Staubli VAL3: page_editTraj.pjx

--- page_editTraj.pjx ---
Parameters version=s7.6.1 stackSize=5000 millimeterUnit=true
Program file=buildList.pgx
Program file=changePoint.pgx
Program file=goTo.pgx
Program file=insertInstr.pgx
Program file=listAdd.pgx
Program file=loadEditTraj.pgx
Program file=loadPage.pgx
Program file=main.pgx
Program file=onBackEvent.pgx
Program file=onEnterEvent.pgx
Program file=onExit.pgx
Program file=onF1Event.pgx
Program file=onF2Event.pgx
Program file=onF3Event.pgx
Program file=onF4Event.pgx
Program file=onF5Event.pgx
Program file=onF6Event.pgx
Program file=onF7Event.pgx
Program file=onF8Event.pgx
Program file=onSpaceEvent.pgx
Program file=onStart.pgx
Program file=refresh.pgx
Program file=refreshDynamic.pgx
Program file=refreshStatic.pgx
Program file=saveIt.pgx
Program file=selectItem.pgx
Program file=setAllAccel.pgx
Program file=setAllBlend.pgx
Program file=setAllSpeed.pgx
Program file=showPoint.pgx
Program file=showStatus.pgx
Program file=unSelectItem.pgx
Data file=page_editTraj.dtx
Library alias=use path=Disk://kernel/userPage/userPage.pjx
Library alias=language path=Disk://kernel/language/language.pjx
Library alias=saveData path=Disk://saveData/saveData.pjx
Library alias=trajType path=Disk://..//templates/trajectory/trajectory.pjx
Library alias=events path=Disk://..//templates/instruction/instruction.pjx
Library alias=tcp path=Disk://kernel/tool/tool.pjx
Library alias=page path=Disk://kernel/template/page/page.pjx
Library alias=cycleStatus path=Disk://cycleStatus/cycleStatus.pjx
Library alias=saveInOut path=Disk://saveInputOutput/saveInputOutput.pjx
Type name=TrajectoryItem path=Disk://kernel/template/TrajectoryItem/TrajectoryItem.pjx
Type name=InstrItem path=Disk://kernel/template/InstrItem/InstrItem.pjx
Type name=FrameItem path=Disk://kernel/template/FrameItem/FrameItem.pjx

--- page_editTraj.dtx ---
bool bButton[8]
  [0] = true
  [1] = true
  [2] = true
  [4] = true
  [5] = true
  [6] = true
  [7] = true
bool bExit
bool bLarge
bool bShowStatus
bool bTrigger
num nClockStatus = 962.397
num nIndex
num nIndexItem
num nKey
num nOldIndex
public num nPage
num nRefresh = 1149.353
num nSelected = -1
num nTime = 1
num nUserItem = 6
num nView
string sAction[3]
string sEvent = "Name: > appro"
public string sItems = "pick"
string sList[17]
  [0] = "Name: > appro"
  [1] = "appro   X > 0   "
  [2] = "appro   Y > 0   "
  [3] = "appro   Z > -50   "
  [4] = "appro  RX > 0   "
  [5] = "appro  RY > 0   "
  [6] = "appro  RZ > 0   "
  [7] = "MoveType > Linear"
  [8] = "Speed    > 1000 mm/s"
  [9] = "Accelerat> 100 %"
  [10] = "Stop  [ ]> "
  [11] = "Blend [x]> 30 mm"
  [12] = "Tool  [ ]>    "
  [13] = "Action1>  "
  [14] = "Action2>  "
  [15] = "Action3>  "
  [16] = "Anticipation > 0 mm"
string sListUser[6]
  [0] = "appro   X > 0   "
  [1] = "appro   Y > 0   "
  [2] = "appro   Z > -50   "
  [3] = "appro  RX > 0   "
  [4] = "appro  RY > 0   "
  [5] = "appro  RZ > 0   "
string sMenu[8]
  [0] = "Here"
  [1] = "Align"
  [2] = "Tool"
  [4] = "Motion"
  [5] = "Delete"
  [6] = "Insert"
  [7] = "Save"
string sMenu8[8]
string sMenuUser[8]
  [0] = "Here"
  [1] = "Align"
  [2] = "Tool"
string sMessage[2]
  [0] = "ON"
  [1] = "OFF"
string sOldListUser
string sTrajName = "pick"
frame fFather = {fatherId=world[0]}

--- main.pgx ---
public program main()
  local bool l_bSave
  local bool l_bOverRide
  local num l_nSize
  local bool l_bUnreached
  local string l_sMessage
begin
  // INIT
  call onStart()
  // LOOP UNTIL nKey=255
  do
    // GOTO
    call goTo(nIndexItem,l_bUnreached)
    if l_bUnreached
      // show the message out of range
      call language:message(l_sMessage,-5)
      call use:timerDialog(l_sMessage,1)
      l_bUnreached=false
    endIf
    //
    call refresh()
    nKey=getKey()
    call use:listevent(nKey,nIndex,sEvent)
    nView=use:nView
    // get Size
    call trajType:getSizeItem(false,l_nSize)
    //
    // OVERRIDE NORMAL FUNCTIONALITY-> POLYMORPHISM
    //
    if nKey>=271 and nKey<=278
      if sMenuUser[nKey-271]!=""
        call trajType:onFunctionEdit(nIndexItem,sEvent,nKey)
        l_bOverRide=true
        l_bSave=true
        call buildList()
      endIf
    endIf
    //
    // OVERRIDE ON ENTER EVENT -> POLYMORPHISM
    //
    if !l_bOverRide
      switch nKey
        case 264
          // left
          if nIndexItem>0
            nIndexItem=nIndexItem-1
            call buildList()
          endIf
        break
        case 268
          // right
          if nIndexItem<(l_nSize-1)
            nIndexItem=nIndexItem+1
            call buildList()
          endIf
        break
        case 259
          // TAB
          bLarge=!bLarge
          call use:setView(bLarge)
        break
        case 32
          call onSpaceEvent(l_bSave)
        break
        case 263
          call onBackEvent(l_bSave)
        break
        case 271
          call onF1Event()
        break
        case 272
          call onF2Event()
        break
        case 273
          call onF3Event()
        break
        case 274
          // Blend
          call onF4Event(l_bSave)
        break
        case 275
          // Speed
          call onF5Event(l_bSave)
        break
        case 276
          // Delete
          call onF6Event(l_bSave)
        break
        case 277
          // Insert
          call onF7Event(l_bSave)
        break
        case 278
          // SAVE
          call onF8Event(l_bSave)
        break
        case 270
          // GO EDIT POINT
          call onEnterEvent(l_bSave)
        break
      endSwitch
    endIf
    l_bOverRide=false
    if nKey==255
      // on Exit
      call onExit(l_bSave)
    endIf
    // release
    delay(0)
  until bExit
  // reset the bit
  bExit=false
end

--- buildList.pgx ---
program buildList()
  local num l_nSize
  local num i
  local string l_sInstruction
  local string l_sMessage
  local string l_sTemp
  local string l_sEmpty
  local TrajectoryItem l_tTraj
  local string l_sData
  local string l_sType
begin
  // INIT the list
  l_sEmpty=""
  call use:stringCopy(l_sEmpty,sList)
  // get all the field
  call trajType:getSizeItem(false,l_nSize)
  call trajType:getTrajItem(l_tTraj,nIndexItem)
  //
  // make the list
  //
  // the name
  call language:message(l_sMessage,21)
  call listAdd(l_sMessage+"> "+l_tTraj.comment)
  if find(l_tTraj.comment,"@")==-1
    // insert the user function if NOT @LINK
    call trajType:getListItem(sListUser,nIndexItem)
    if sListUser!=""
      for i=0 to size(sListUser)-1
        call listAdd(sListUser[i])
      endFor
      nUserItem=size(sListUser)
    else
      nUserItem=0
    endIf
    // check the size for the line underline
    if size(sListUser)!=size(sOldListUser) and sOldListUser!=""
      nSelected=nIndex+(size(sListUser)-size(sOldListUser))
      // copy it
      call use:stringCopy(sListUser,sOldListUser)
      use:bUseRefresh=true
    else
      nSelected=-1
    endIf
  else
    // empty it
    call use:stringCopy(l_sEmpty,sListUser)
    nUserItem=0
    nSelected=nIndex
  endIf
  // the movetype
  switch l_tTraj.moveType
    case 0
      // JOINT
      call language:message(l_sTemp,164)
      call language:message(l_sMessage,157)
      call use:strfill(l_sMessage,9,l_sMessage)
      call listAdd(l_sMessage+"> "+l_sTemp)
      call language:message(l_sMessage,158)
      call use:strfill(l_sMessage,9,l_sMessage)
      call listAdd(l_sMessage+"> "+toString("",l_tTraj.nom_speed.vel)+" %")
    break
    case 1
      //LINEAR
      call language:message(l_sTemp,165)
      call language:message(l_sMessage,157)
      call use:strfill(l_sMessage,9,l_sMessage)
      call listAdd(l_sMessage+"> "+l_sTemp)
      call language:message(l_sMessage,158)
      call use:strfill(l_sMessage,9,l_sMessage)
      call listAdd(l_sMessage+"> "+toString("",l_tTraj.nom_speed.tvel)+" mm/s")
    break
    case 2
      //  CIRCULAR
      call language:message(l_sTemp,166)
      call language:message(l_sMessage,157)
      call use:strfill(l_sMessage,9,l_sMessage)
      call listAdd(l_sMessage+"> "+l_sTemp)
      call language:message(l_sMessage,158)
      call use:strfill(l_sMessage,9,l_sMessage)
      call listAdd(l_sMessage+"> "+toString("",l_tTraj.nom_speed.tvel)+" mm/s")
    break
  endSwitch
  // ACCELERATION
  call language:message(l_sMessage,159)
  call use:strfill(l_sMessage,9,l_sMessage)
  call listAdd(l_sMessage+"> "+toString("",l_tTraj.nom_speed.accel)+" %")
  // STOP
  call use:showBoolStatus(l_tTraj.toStop,l_sTemp)
  call language:message(l_sMessage,174)
  call use:strfill(l_sMessage,6,l_sMessage)
  l_sMessage=l_sMessage+l_sTemp
  if l_tTraj.toStop
    // STOP
    if round(l_tTraj.nStop)!=l_tTraj.nStop
      l_sTemp=toString(".2",l_tTraj.nStop)+" sec"
    else
      l_sTemp=toString("",l_tTraj.nStop)+" sec"
    endIf
  else
    // NO STOP
    l_sTemp=""
  endIf
  call listAdd(l_sMessage+"> "+l_sTemp)
  // BLEND
  if l_tTraj.nom_speed.blend==off
    l_sTemp="[ ]> "
  else
    if l_tTraj.nom_speed.blend==joint
      l_sTemp="[x]> "+toString("",l_tTraj.nom_speed.leave)+" mm"
    endIf
  endIf
  call language:message(l_sMessage,175)
  call use:strfill(l_sMessage,6,l_sMessage)
  call listAdd(l_sMessage+l_sTemp)
  // TCP ON OFF
  call language:message(l_sMessage,123)
  call use:strfill(l_sMessage,6,l_sMessage)
  switch l_tTraj.nTcpAction
    case 1
      l_sTemp="[x]> ON "
    break
    case 2
      l_sTemp="[x]> OFF"
    break
    default
      l_sTemp="[ ]>    "
    break
  endSwitch
  call listAdd(l_sMessage+l_sTemp)
  // INSTRUCTION
  call language:message(l_sMessage,176)
  // copy all
  for i=0 to size(l_tTraj.iInstr)-1
    l_sData=l_tTraj.iInstr[i].sData
    l_sType=l_tTraj.iInstr[i].sType
    call saveInOut:replaceIO(l_sData,l_sType,l_sData)
    call listAdd(l_sMessage+toString("1",i+1)+"> "+l_sType+" "+l_sData)
  endFor
  // DISTANCE
  call language:message(l_sMessage,177)
  call listAdd(l_sMessage+" > "+toString("",l_tTraj.distance)+" mm")
  // update
  use:bUseRefresh=true
end

--- changePoint.pgx ---
program changePoint(num x_nIndex)
  local num i
  local string l_sMessage[3]
  local num l_nLocal
  local bool l_bOk
  local num l_nStop
  local string l_sButton[2]
  local string l_sEmpty
  local TrajectoryItem l_tTraj
  local InstrItem l_iInstr
  local string l_sItem
  local string l_sData
  local string l_sPath
begin
  //
  // Init and save the right side of the string starting from ">"
  //
  logMsg("[KERNEL] INTERFACE:Change Point: "+sEvent+" item: "+toString("",nIndexItem))
  //i=find(sEvent,">")+1
  call use:findPos(sEvent,">",i)
  i=i+1
  //
  if i!=-1
    //
    //  There are 10 fields,
    //
    call trajType:getTrajItem(l_tTraj,nIndexItem)
    // clean the line
    call use:listcursor(use:nView,false)
    l_sEmpty=""
    switch x_nIndex
      case 0
        //
        //  comment for the point
        //
        // read the name
        call use:read(i+40-use:nBottomX,use:nView+1,l_tTraj.comment,10,false)
      break
      case 1
        //
        //  change the movetype (0->Joint, 1->Linear, 2->Circle)
        //
        // JOINT
        if trajType:bMoveType[0]
          // normaly with joint can be also linear and circle
          call language:message(l_sMessage,164)
          call language:message(l_sMessage[1],165)
          call language:message(l_sMessage[2],166)
          if trajType:bMoveType[1]
            l_sMessage=l_sMessage+","+l_sMessage[1]
          endIf
          if trajType:bMoveType[2] and nIndexItem!=0
            l_sMessage=l_sMessage+","+l_sMessage[2]
          endIf
        else
          // only linear
          if trajType:bMoveType[1]
            l_sMessage=l_sMessage
          endIf
        endIf
        // compose the string
        call use:stringToArray(l_sMessage,sMessage)
        // look for multiple istance
        if size(sMessage)>1
          //
          l_nLocal=l_tTraj.moveType
          call use:changeValue(l_tTraj.moveType,0,0,i+40-use:nBottomX,use:nView+1,sMessage)
          if l_nLocal!=l_tTraj.moveType
            switch l_tTraj.moveType
              case 0
                if l_tTraj.nom_speed.tvel!=9999
                  l_tTraj.nom_speed.vel=(l_tTraj.nom_speed.tvel)/15
                  l_tTraj.nom_speed.tvel=9999
                endIf
              break
              case 1,2
                if l_tTraj.nom_speed.vel<450
                  l_tTraj.nom_speed.tvel=(l_tTraj.nom_speed.vel)*15
                  l_tTraj.nom_speed.vel=450
                endIf
              break
            endSwitch
            // update the line
            if l_nLocal==2 and nIndex>0 and nView>0
              // refresh the cursor
              nView=nView-1
              nIndex=nIndex-1
            else
              if l_tTraj.moveType==2
                // refresh the cursor
                nView=nView+1
                nIndex=nIndex+1
              endIf
            endIf
          endIf
        endIf
      break
      case 2
        //
        //  change the speed
        //
        if l_tTraj.moveType==0
          call use:changeValue(l_tTraj.nom_speed.vel,1,400,i+40-use:nBottomX,use:nView+1,l_sEmpty)
        else
          if l_tTraj.moveType==1 or l_tTraj.moveType==2
            call use:changeValue(l_tTraj.nom_speed.tvel,1,6000,i+40-use:nBottomX,use:nView+1,l_sEmpty)
          endIf
        endIf
      break
      case 3
        //
        //  change the acceleration
        //
        call use:changeValue(l_tTraj.nom_speed.accel,1,800,i+40-use:nBottomX,use:nView+1,l_sEmpty)
        l_tTraj.nom_speed.decel=l_tTraj.nom_speed.accel
      break
      case 4
        //
        //  put a stop, after the robot reach to the point
        //
        l_nLocal=l_tTraj.nStop
        call use:changeValue(l_nLocal,-1,100,i+40-use:nBottomX,use:nView+1,l_sEmpty)
        //
        if l_nLocal<0
          // no stop
          l_tTraj.toStop=false
          l_tTraj.nStop=0
        else
          // stop using time
          l_tTraj.toStop=true
          l_tTraj.nStop=l_nLocal
        endIf
      break
      case 5
        //
        //  set the blend (joint/off) for the point
        //
        l_nLocal=l_tTraj.nom_speed.leave
        call use:changeValue(l_nLocal,-1,400,i+40-use:nBottomX,use:nView+1,l_sEmpty)
        if l_nLocal<0
          l_tTraj.nom_speed.blend=off
        else
          l_tTraj.nom_speed.leave=l_tTraj.nom_speed.reach=l_nLocal
          l_tTraj.nom_speed.blend=joint
        endIf
      break
      case 6
        //
        // set TCP ON/OFF
        //
        // NB: 0>NONE 1>ON 2>OFF
        call use:stringToArray("ON,OFF",sMessage)
        if l_tTraj.nTcpAction!=0 and abs(l_tTraj.nTcpAction)<3
          // NOTE
          // use only absolute
          l_tTraj.nTcpAction=abs(l_tTraj.nTcpAction)-1
        else
          l_tTraj.nTcpAction=0
        endIf
        call use:changeValue(l_tTraj.nTcpAction,0,0,i+40-use:nBottomX,use:nView+1,sMessage)
        // give back increase by one
        l_tTraj.nTcpAction=l_tTraj.nTcpAction+1
      break
      case 7,8,9
        //
        //  Insert the instruction
        //
        // insert a new one
        if l_tTraj.iInstr[x_nIndex-7].sType!=""
          // show it
          if l_tTraj.iInstr[x_nIndex-7].sType=="OUT" or l_tTraj.iInstr[x_nIndex-7].sType=="IN" or l_tTraj.iInstr[x_nIndex-7].sType=="EMAP"
            popUpMsg(l_tTraj.iInstr[x_nIndex-7].sType+" "+l_tTraj.iInstr[x_nIndex-7].sData)
          else
            // update
            l_sItem=l_tTraj.iInstr[x_nIndex-7].sType
            l_sData=l_tTraj.iInstr[x_nIndex-7].sData
            call saveData:getPathInstr(l_sItem,l_sPath)
            events:libLoad(l_sPath)
            delay(0)
            call events:onEdit(l_sData)
            if l_sData!=""
              l_tTraj.iInstr[x_nIndex-7].sData=l_sData
            endIf
          endIf
        else
          // insert
          call insertInstr(l_iInstr)
          if l_iInstr.sData!=""
            l_tTraj.iInstr[x_nIndex-7]=l_iInstr
          endIf
        endIf
      break
      case 10
        //
        //  set the distance from the point where the call will be actived
        //
        call use:changeValue(l_tTraj.distance,-300,300,i+40-use:nBottomX,use:nView+1,l_sEmpty)
      break
    endSwitch
    //set and exit
    call trajType:setTrajItem(l_tTraj,nIndexItem)
  endIf
  //
  call use:nullKey(nKey)
end

--- goTo.pgx ---
program goTo(num x_nIndex, bool& x_bUnreached[])
  local bool l_bUnreached
  local num l_nIndexTool
  local tool l_tTool
  local TrajectoryItem l_tTraj
begin
//  if !cycleStatus:bCycle
//    if cycleStatus:nWorkingMode==1 and isPowered()
//      // check for the index
//      if nOldIndex!=x_nIndex or (cycleStatus:nWorkingStatus!=0 and cycleStatus:nWorkingStatus!=6)
//        if !isEmpty()
//          resetMotion()
//        endIf
//        if nOldIndex!=x_nIndex
//          nOldIndex=x_nIndex
//        endIf
//      else
//        if isEmpty() and cycleStatus:nWorkingStatus==0
//          // get the data to move
//          call trajType:getTool(l_nIndexTool)
//          call tcp:getTool(l_tTool,l_nIndexTool)
//          call trajType:getTrajItem(l_tTraj,x_nIndex)
//          //
//          // use a sTemp mdesc to set the blend off
//          //
//          l_tTraj.nom_speed.blend=off
//          call trajType:goTo(l_tTool,l_tTraj.nom_speed,l_tTraj.moveType,x_bUnreached,x_nIndex)
//          call showPoint()
//        endIf
//      endIf
//    else
//      if cycleStatus:nWorkingMode!=1
//        resetMotion()
//      endIf
//    endIf
//  endIf
end

--- insertInstr.pgx ---
program insertInstr(InstrItem& x_iInstr[])
  local num i
  local string l_sMessage
  local num l_nIndex
  local string l_sItem
  local string l_sPath
begin
  // create the list
  call use:setSizeList(15,0,15,11)
  call use:setView(false)
  call language:message(l_sMessage,35)
  call use:listcreate(l_sMessage)
  // insert the action on Point
  call use:listadd(saveData:sInstrOnPoint)
  call use:listupdate(0)
  // SELECT THE ITEM
  x_iInstr.sData=""
  do
    i=get()
    l_nIndex=0
    call use:listevent(i,l_nIndex,l_sItem)
  until i==255 or i==270
  // update
  x_iInstr.sType=l_sItem
  // update
  call saveData:getPathInstr(l_sItem,l_sPath)
  if l_sItem!="" and i==270
    events:libLoad(l_sPath)
    delay(0)
    call events:onInsert(l_sItem)
    x_iInstr.sData=l_sItem
  endIf
end

--- loadEditTraj.pgx ---
program loadEditTraj(string x_sName)
  local num i
  local num l_nIndex
  local string l_sPath
begin
  // load the traj type
  call saveData:getPathInstr(saveData:sTrajTypeUsing,l_sPath)
  i=trajType:libLoad(l_sPath)
  delay(0)
  if i!=0
    popUpMsg("error load traj type on START "+saveData:sTrajTypeUsing+toString("",i))
  endIf
  // save the name
  sTrajName=x_sName
end

--- loadPage.pgx ---
program loadPage(string x_sPage, string& x_sItems[])
// load the next page
  local num i
  local string l_sMessage
begin
  // look if the page libload is correct
  i=page:libLoad(x_sPage)
  delay(0)
  if i!=0
    logMsg("[KERNEL] INTERFACE:PAGE LIBLOAD "+x_sPage+" result "+toString("",i))
    call language:message(l_sMessage,-7)
    popUpMsg(l_sMessage+x_sPage+" ; "+toString("",i))
  else
    // copy all the field from x_sItems to the next page
    call use:stringCopy(x_sItems,page:sItems)
    call page:main()
    // copy BACK
    call use:stringCopy(page:sItems,x_sItems)
  endIf
end

--- onBackEvent.pgx ---
program onBackEvent(bool& x_bSave[] (dimensions=1))
  local num i
  local string l_sMessage[3]
  local num l_nLocal
  local bool l_bYes
  local string l_sAction[3]
  local num l_nIndex
  local string l_sButton[2]
  local TrajectoryItem l_tTraj
begin
  //
  // NB sEvent is the selected
  // element in the LIST
  //
  if nIndex!=0
    l_nIndex=nIndex-nUserItem
  else
    // change the name
    call changePoint(0)
  endIf
  if (l_nIndex)>0
    //
    //  There are 7 fields,
    //
    //
    call trajType:getTrajItem(l_tTraj,nIndexItem)
    switch l_nIndex
      case 1
        //
        //  change the movetype
        //
      break
      case 2
        //
        //  change the speed
        //
      break
      case 3
        //
        //  change the acceleration
        //
      break
      case 4
        //
        //  put a stop, after the robot reach to the point
        //
        // CLEAR THE STOP
        l_tTraj.toStop=false
      break
      case 5
        //
        //  set the blend (joint/off) for the point
        //
        l_tTraj.nom_speed.blend=off
      break
      case 6
        //
        // set TCP ON/OFF
        //
        // SET TCP OFF
        l_tTraj.nTcpAction=0
      break
      case 7,8,9
        //
        //  Delete the instruction
        //
        if l_tTraj.iInstr[l_nIndex-7].sType!=""
          call language:message(l_sMessage,171)
          call language:getYesNo(l_sButton)
          // ask the yes_no question
          call use:yes_no(l_sMessage,l_sButton,l_bYes)
          if l_bYes
            l_tTraj.iInstr[l_nIndex-7].sType=""
            l_tTraj.iInstr[l_nIndex-7].sData=""
          endIf
        endIf
      break
      case 10
        //
        //  set the distance from the point where the call will be actived
        //
        l_tTraj.distance=0
      break
    endSwitch
    //set and exit
    x_bSave=true
    call trajType:setTrajItem(l_tTraj,nIndexItem)
    call buildList()
  endIf
end

--- onEnterEvent.pgx ---
program onEnterEvent(bool& x_bSave (dimensions=1))
begin
  //
  // NB sEvent is the selected
  // element in the LIST
  //
  if nIndex==0
    // change the name
    call changePoint(0)
  else
    if (nIndex-nUserItem)>0
      // change the default value
      call changePoint(nIndex-nUserItem)
      x_bSave=true
    else
      // change the custom item
      call trajType:onEditItem(sEvent,nIndex-1,nIndexItem)
    endIf
  endIf
  x_bSave=true
  call buildList()
end

--- onExit.pgx ---
program onExit(bool& x_bSave[] (dimensions=1))
  local string l_sMessage
  local bool l_bYes
  local bool l_bCancel
  local string l_sButton[2]
begin
  // saveIt
  if x_bSave
    call language:message(l_sMessage,-1)
    call language:getYesNo(l_sButton)
    // ask the yes_no question
    call use:yes_no_cancel(l_sMessage,l_sButton,l_bYes,l_bCancel)
    if l_bYes
      call saveIt(x_bSave)
    endIf
    // look for the cancel button
    bExit=!l_bCancel
  else
    // exit frome the page
    bExit=true
  endIf
  // send Back
  if size(sItems)>1
    sItems[1]=toString("",nIndexItem)
  endIf
  // null key
  call use:nullKey(nKey)
  // reset the show status
  bShowStatus=false
  // resetMotion
  if !cycleStatus:bCycle
    resetMotion()
  endIf
end

--- onF1Event.pgx ---
program onF1Event()
begin
  // look if the bButton is enable
  if bButton[0]
    //
  endIf
end

--- onF4Event.pgx ---
program onF4Event(bool& x_bSave[] (dimensions=1))
  local string l_sMessage
  local num l_nActual
  local num l_nOldValue
  local num l_nX
  local num l_nY
begin
  // look if the bButton is enable
  if bButton[3]
    //
    //
    //
  endIf
end

--- onF5Event.pgx ---
program onF5Event(bool& x_bSave[])
  local string l_sMessage
  local num l_nActual
  local num l_nOldValue
  local num l_nMoveType
  local num l_nIndex
  local num l_nKey
  local string l_sEvent
  local TrajectoryItem l_tTraj
begin
  // look if the bButton is enable
  if bButton[4]
    //
    // build a little List to select speed accel blend
    //
    call use:clear(0,13)
    call use:type(21,13,sMenu[4])
    call use:setSizeList(17,8,12,3)
    call use:listcreate("")
    // speed
    call language:message(l_sMessage,158)
    call use:listadd(l_sMessage)
    // accel
    call language:message(l_sMessage,159)
    call use:listadd(l_sMessage)
    // blend
    call language:message(l_sMessage,175)
    call use:listadd(l_sMessage)
    //
    call use:listupdate(0)
    do
      l_nKey=get()
      call use:listevent(l_nKey,l_nIndex,l_sEvent)
    until l_nKey==270 or l_nKey==255
    if l_nKey==270
      // get the traj Item
      call trajType:getTrajItem(l_tTraj,nIndexItem)
      // switch case
      switch l_nIndex
        case 0
          //
          // change the speed
          //
          call language:message(l_sMessage,161)
          switch l_tTraj.moveType
            case 0
              // JOINT
              l_nActual=l_nOldValue=l_tTraj.nom_speed.vel
              call use:insertDialog(l_sMessage+" %",l_nActual,1,400)
            break
            case 1,2
              //LINEAR CIRCULAR
              l_nActual=l_nOldValue=l_tTraj.nom_speed.tvel
              call use:insertDialog(l_sMessage+" mm/sec ",l_nActual,1,6000)
            break
          endSwitch
          call setAllSpeed(l_nActual,l_nOldValue)
          logMsg("[VALTRAJ] INTERFACE:Change all speed from: "+toString("",l_nOldValue)+" to: "+toString("",l_nActual))
        break
        case 1
          //
          // CHANGE ALL THE ACCEL
          //
          call language:message(l_sMessage,162)
          l_nActual=l_nOldValue=l_tTraj.nom_speed.accel
          call use:insertDialog(l_sMessage,l_nActual,1,800)
          call setAllAccel(l_nActual,l_nOldValue)
          logMsg("[VALTRAJ] INTERFACE:Change all accel from: "+toString("",l_nOldValue)+" to: "+toString("",l_nActual))
        break
        case 2
          //
          // CHANGE ALL THE BLEND
          //
          call language:message(l_sMessage,178)
          l_nActual=l_nOldValue=l_tTraj.nom_speed.leave
          call use:insertDialog(l_sMessage,l_nActual,-1,400)
          call setAllBlend(l_nActual,l_nOldValue)
          logMsg("[VALTRAJ] INTERFACE:Change all blend from: "+toString("",l_nOldValue)+" to: "+toString("",l_nActual))
        break
      endSwitch
      // save and return
      x_bSave=true
      call buildList()
    endIf
  endIf
end

--- onF6Event.pgx ---
program onF6Event(bool& x_bSave[])
  local string l_sMessage
  local bool l_bYes
  local num l_nSize
  local num l_nFound
  local string l_sEvent
  local string l_sButton[2]
  local num l_nItem
begin
  // look if the bButton is enable
  if bButton[5]
    //
    // DELETE
    //
    call language:message(l_sMessage,80)
    call language:getYesNo(l_sButton)
    // ask the yes_no question
    call use:yes_no(l_sMessage,l_sButton,l_bYes)
    if l_bYes
      l_nItem=nIndexItem
      call trajType:getSizeItem(false,l_nSize)
      if l_nSize>1
        call trajType:deleteItem(nIndexItem)
        if nIndexItem>0
          nIndexItem=nIndexItem-1
        else
          nIndexItem=l_nItem
        endIf
        //refresh
        call buildList()
        use:bUseRefresh=true
      endIf
    endIf
    x_bSave=true
  endIf
end

--- onF7Event.pgx ---
program onF7Event(bool& x_bSave[] (dimensions=1))
  local TrajectoryItem l_tTraj
  local num l_nItem
begin
  // look if the bButton is enable
  if bButton[6]
    //
    // insert
    l_nItem=nIndexItem
    // insert the default value
    call trajType:insertItem(nIndexItem,nIndexItem+1)
    call trajType:getTrajItem(l_tTraj,nIndexItem)
    l_tTraj.comment=""
    l_tTraj.toStop=false
    call trajType:setTrajItem(l_tTraj,nIndexItem+1)
    nIndexItem=nIndexItem+1
    // rebuild list
    call buildList()
    x_bSave=true
    //refresh
    call buildList()
    use:bUseRefresh=true
  endIf
end

--- onF8Event.pgx ---
program onF8Event(bool& x_bSave[] (dimensions=1))
  local num i
begin
  // look if the bButton is enable
  if bButton[7]
    //
    call saveIt(x_bSave)
  endIf
end

--- onSpaceEvent.pgx ---
program onSpaceEvent(bool& x_bSave[])
  local num i
  local string l_sMessage[3]
  local num l_nLocal
  local bool l_bYes
  local string l_sAction[3]
  local num l_nIndex
  local TrajectoryItem l_tTraj
  local bool l_bStop
begin
  //
  // NB sEvent is the selected
  // element in the LIST
  //
  l_nIndex=nIndex-nUserItem
  if (nIndex-nUserItem)>0
    //
    //  There are 7 fields,
    //
    //
    call trajType:getTrajItem(l_tTraj,nIndexItem)
    switch l_nIndex
      case 0
        //
        //  comment for the point
        //
      break
      case 1
        //
        //  change the movetype
        //
      break
      case 2
        //
        //  change the speed
        //
      break
      case 3
        //
        //  change the acceleration
        //
      break
      case 4
        //
        //  put a stop, after the robot reach to the point
        //
        l_tTraj.toStop=!l_tTraj.toStop
      break
      case 5
        //
        //  set the blend (joint/off) for the point
        //
        if l_tTraj.nom_speed.blend==off
          l_tTraj.nom_speed.blend=joint
        else
          l_tTraj.nom_speed.blend=off
        endIf
      break
      case 6
        //
        // set TCP ON/OFF
        //
        if l_tTraj.nTcpAction!=0
          l_tTraj.nTcpAction=-l_tTraj.nTcpAction
        else
          // ON by default
          l_tTraj.nTcpAction=1
        endIf
      break
      case 7,8,9
        //
        //  Insert the instruction
        //
      break
      case 10
        //
        //  set the distance from the point where the call will be actived
        //
      break
    endSwitch
    //set and exit
    call trajType:setTrajItem(l_tTraj,nIndexItem)
    x_bSave=true
    call buildList()
  endIf
end

--- onStart.pgx ---
program onStart()
  local num i
  local num l_nIndex
  local bool l_bOk
begin
  // INIT
  sTrajName=sItems
  nView=0
  nIndex=0
  bExit=false
  link(fFather,world)
  call trajType:getFrame(fFather,false)
  // set the index
  l_bOk=true
  if size(sItems)>1 and sItems[1]!=""
    toNum(sItems[1],nIndexItem,l_bOk)
  else
    nIndexItem=0
  endIf
  // empty the userMenu
  for i=0 to size(sMenuUser)-1
    sMenuUser[i]=""
  endFor
  // load the traj type
  call loadEditTraj(sItems)
  //endIf
  //
  // logMsg
  logMsg("[KERNEL] INTERFACE:PAGE Edit TRAJ")
  // reset the Key pressure
  call use:nullKey(nKey)
  // define the list
  call buildList()
  //
end

--- refresh.pgx ---
program refresh()
// // page refresh
begin
  if !use:bShowDialog and !cycleStatus:bShowMessage
    //
    // refresh the static message
    if (nKey>=270 and nKey<=278) or (nKey==264 or nKey==268) or (use:bUseRefresh and !bShowStatus)
      call refreshStatic()
      call refreshDynamic()
    else
      if !bShowStatus
        // refresh the Dynamic message
        if abs(clock()-nRefresh)>nTime
          call refreshDynamic()
        endIf
      endIf
    endIf
  endIf
  //
  call showStatus()
end

--- refreshDynamic.pgx ---
program refreshDynamic()
begin
  // DO NOT CHANGE
  nRefresh=clock()
  use:bUseRefresh=false
  call showPoint()
  //
  // ADD HERE
  //
end

--- refreshStatic.pgx ---
program refreshStatic()
  local string l_sMenu
  local num i
  local string l_sInstruction
  local num l_nSize
  local string l_sMessage
  local mdesc l_mDesc
  local num l_nTcpAction
  local string l_sName
  local string l_sEmpty
  local bool l_bStop
  local num l_nEmpty
  local num l_nIndexTool
  local TrajectoryItem l_tTraj
  local string l_sType
  local string l_sData
begin
  cls()
  //
  // set the view of the page..
  //
  // SET THE PAGE NUMBER
  use:nPage=100000
  // USE <>PROFILE for <>PAGE
  use:nPage=use:nPage+abs(limit(saveData:mode,0,2)-2)
  // load the menu page
  if saveData:language!="japanese"
    // SET THE VIEW OF THE PAGE
    call language:page(l_sMessage,use:nPage)
    // define the menu
    call use:stringToArray(l_sMessage,sMenu)
  else
    // japanese use the array for the menu
    call language:page(sMenu8,use:nPage)
    call use:stringCopy(sMenu8,sMenu)
  endIf
  //
  // polymorphism
  //
  // get the user Menu or special one
  call trajType:getFunctionEdit(sMenuUser)
  // OVERRIDE
  for i=0 to size(sMenuUser)-1
    if sMenuUser[i]!=""
      sMenu[i]=sMenuUser[i]
    endIf
  endFor
  // check for the here if not in cycle
  if cycleStatus:bCycle or cycleStatus:bSimulation
    sMenu[0]=""
  endIf
  // remove the insert delete in this page
  sMenu[5]=sMenu[6]=""
  if saveData:language!="japanese"
    // set the menu
    call use:setMenu(sMenu,true,3)
  else
    // set the menu
    call use:setMenu(sMenu,false,3)
  endIf
  call use:getMenu(sMenu,bButton)
  //
  // CREATE THE LIST
  //
  // define your list size for default
  // get the nSize
  call trajType:getSizeItem(false,l_nSize)
  call use:setSizeList(19,0,19,10)
  call use:setView(bLarge)
  // show the title...
  l_sName=sTrajName
  if !bLarge and len(sTrajName)>12
    // as japanese told us
    l_sName=left(sTrajName,9)+"¬"+right(sTrajName,2)
  endIf
  call use:listcreate(l_sName+" "+toString("3",nIndexItem+1)+"/"+toString("3",l_nSize))
  //
  call use:listadd(sList)
  //
  // refresh the cursor
  use:nView=nView
  // refresh the list
  call use:selectNewField(nSelected,nIndex,nView)
  // show the instruction
  l_sEmpty=""
  l_bStop=false
  l_nEmpty=0
  call trajType:getTrajItem(l_tTraj,nIndexItem)
  // select the action
  switch l_tTraj.nTcpAction
    case 1
      l_sInstruction="[ON],"
    break
    case 2
      l_sInstruction="[OFF],"
    break
    default
    break
  endSwitch
  l_sType=l_tTraj.iInstr[0].sType
  l_sData=l_tTraj.iInstr[0].sData
  call saveInOut:replaceIO(l_sData,l_sType,l_sData)
  l_sInstruction=l_sInstruction+l_sType+" "+l_sData
  for i=1 to size(l_tTraj.iInstr)-1
    if l_tTraj.iInstr[i].sType!=""
      l_sType=l_tTraj.iInstr[i].sType
      l_sData=l_tTraj.iInstr[i].sData
      call saveInOut:replaceIO(l_sData,l_sType,l_sData)
      l_sInstruction=l_sInstruction+","+l_sType+" "+l_sData
    endIf
  endFor
  call use:typeLen(0,12,l_sInstruction,40)
  // TOOL - FRAME
  if !bLarge
    call trajType:getTool(i)
    call language:message(l_sMessage,124)
    call tcp:getName(l_sName,i)
    call use:type(0,0,l_sMessage+":"+toString("",i)+" "+l_sName)
    call trajType:getFrameId(i)
    call language:message(l_sMessage,124)
    l_sName=saveData:fFrameItem[i].sName
    call use:type(0,1,"Frame:"+toString("",i)+" "+l_sName)
  endIf
end

--- saveIt.pgx ---
program saveIt(bool& x_bSave[] (dimensions=1))
  local string l_sMessage
  local num l_nResult
  local string l_sResult
begin
  // unselect ALL
  call unSelectItem()
  // do the onSave trajtype
  l_sResult=""
  call trajType:onSave(l_sResult)
  //
  if l_nResult==0
    logMsg("[KERNEL] INTERFACE:Save the trajectory "+saveData:sTrajTypeUsing+": "+sTrajName)
    x_bSave=false
    call language:message(l_sMessage,-4)
    call use:timerDialog(l_sMessage,1)
  else
    popUpMsg("Save code error "+toString("",l_nResult))
  endIf
end

--- selectItem.pgx ---
public program selectItem(num x_nIndex (dimensions=1))
  local string l_sItem
  local TrajectoryItem l_tTraj
begin
  //
  // select or unselect one item
  //
  call trajType:getTrajItem(l_tTraj,x_nIndex)
  // check for the selected flag
  if find(l_tTraj.comment,"#")==-1
    l_tTraj.comment="#"+l_tTraj.comment
  else
    l_tTraj.comment=right(l_tTraj.comment,len(l_tTraj.comment)-1)
  endIf
  // set it
  call trajType:setTrajItem(l_tTraj,x_nIndex)
end

--- setAllAccel.pgx ---
public program setAllAccel(num x_nNewValue (dimensions=1), num x_nOldValue (dimensions=1))
  local num i
  local num l_nSize
  local TrajectoryItem l_tTraj
begin
  //
  // change all the accel(equal at newValue)to the newValue
  //
  if x_nNewValue!=x_nOldValue
    call trajType:getSizeItem(false,l_nSize)
    // scan it
    for i=0 to (l_nSize-1)
      // get it
      call trajType:getTrajItem(l_tTraj,i)
      // check if is OK
      if l_tTraj.nom_speed.accel==x_nOldValue
        l_tTraj.nom_speed.accel=l_tTraj.nom_speed.decel=x_nNewValue
      endIf
      // set IT
      call trajType:setTrajItem(l_tTraj,i)
    endFor
  endIf
end

--- setAllBlend.pgx ---
public program setAllBlend(num x_nNewValue, num x_nOldValue)
  local num i
  local num l_nSize
  local TrajectoryItem l_tTraj
begin
  // check if is OK
  if x_nNewValue!=x_nOldValue
    // get the size
    call trajType:getSizeItem(false,l_nSize)
    for i=0 to (l_nSize-1)
      // get it
      call trajType:getTrajItem(l_tTraj,i)
      // check it
      if l_tTraj.nom_speed.leave==x_nOldValue or (l_tTraj.nom_speed.blend==off and x_nOldValue==-1)
        if x_nNewValue<0
          l_tTraj.nom_speed.blend=off
        else
          l_tTraj.nom_speed.leave=l_tTraj.nom_speed.reach=x_nNewValue
          l_tTraj.nom_speed.blend=joint
        endIf
      endIf
      // set it
      call trajType:setTrajItem(l_tTraj,i)
    endFor
  endIf
end

--- setAllSpeed.pgx ---
program setAllSpeed(num x_nNewValue (dimensions=1), num x_nOldValue (dimensions=1))
  local num i
  local num l_nSize
  local TrajectoryItem l_tTraj
begin
  // change all the speed
  if x_nNewValue!=x_nOldValue
    call trajType:getSizeItem(false,l_nSize)
    // scan it
    for i=0 to (l_nSize-1)
      // get the trajitem
      call trajType:getTrajItem(l_tTraj,i)
      // JOINT MOVEMENT
      if (l_tTraj.moveType==0) and (x_nOldValue==l_tTraj.nom_speed.vel)
        l_tTraj.nom_speed.vel=x_nNewValue
        // LINEAR MOVEMENT
      elseIf (l_tTraj.moveType==1 or l_tTraj.moveType==2) and (x_nOldValue==l_tTraj.nom_speed.tvel)
        l_tTraj.nom_speed.tvel=x_nNewValue
      endIf
      // set the trajItem
      call trajType:setTrajItem(l_tTraj,i)
    endFor
  endIf
end

--- showPoint.pgx ---
program showPoint()
  local point l_pPoint[2]
  local num l_nIndexTool
  local tool l_tTool
  local point l_pHere
  local num i
  local joint l_jHere
begin
  // check for the @ position and the ! position
  call trajType:getPoint(l_pPoint,false,nIndexItem)
  call trajType:getTool(l_nIndexTool)
  call tcp:getTool(l_tTool,l_nIndexTool)
  l_pHere=here(l_tTool,fFather)
  if isEmpty() and distance(l_pHere.trsf,position(l_pPoint,fFather))<0.1
    call use:type(use:nTopX,use:nTopY+1,"@")
  elseIf position(l_pPoint,fFather)=={0,0,0,0,0,0}
    call use:type(use:nTopX,use:nTopY+1,"0")
  elseIf distance(position(l_pPoint,fFather),l_pHere.trsf)<10
    call use:type(use:nTopX,use:nTopY+1,"~")
  elseIf !pointToJoint(l_tTool,l_jHere,l_pPoint,l_jHere)
    call use:type(use:nTopX,use:nTopY+1,"!")
  else
    call use:type(use:nTopX,use:nTopY+1,"│")
  endIf
end

--- showStatus.pgx ---
program showStatus()
  local joint l_jHere
  local point l_pHere
  local string l_sMessage[2]
  local tool l_tTool
  local num l_nIndexTool
begin
  //
  // show an dialog box with
  // the current Joint/cartesian position
  //
  call trajType:getTool(l_nIndexTool)
  call tcp:getTool(l_tTool,l_nIndexTool)
  if cycleStatus:nWorkingStatus>1 and cycleStatus:nWorkingStatus<5 and cycleStatus:nWorkingMode==1
    // set a timer of x second then the message disappear ..
    if !bTrigger
      nClockStatus=clock()
      bTrigger=true
      bShowStatus=true
    endIf
    if clock()-nClockStatus<saveData:nTimeDialog
      if cycleStatus:nWorkingStatus==2
        l_jHere=herej()
        l_sMessage="J1:"+toString("7.1",l_jHere.j1)
        l_sMessage=l_sMessage+"  J2:"+toString("7.1",l_jHere.j2)
        l_sMessage=l_sMessage+"  J3:"+toString("7.1",l_jHere.j3)+"#"
        l_sMessage=l_sMessage+"J4:"+toString("7.1",l_jHere.j4)
        l_sMessage=l_sMessage+"  J5:"+toString("7.1",l_jHere.j5)
        l_sMessage=l_sMessage+"  J6:"+toString("7.1",l_jHere.j6)
      else
        l_pHere=here(l_tTool,fFather)
        l_sMessage="X :"+toString("7.1",l_pHere.trsf.x)
        l_sMessage=l_sMessage+"  Y :"+toString("7.1",l_pHere.trsf.y)
        l_sMessage=l_sMessage+"  Z :"+toString("7.1",l_pHere.trsf.z)+"#"
        l_sMessage=l_sMessage+"RX:"+toString("7.1",l_pHere.trsf.rx)
        l_sMessage=l_sMessage+"  RY:"+toString("7.1",l_pHere.trsf.ry)
        l_sMessage=l_sMessage+"  RZ:"+toString("7.1",l_pHere.trsf.rz)
      endIf
      call use:timerDialog(l_sMessage,0)
    else
      // disable it
      bShowStatus=false
    endIf
  else
    // reset it
    if bTrigger and !cycleStatus:bCycle
      resetMotion()
      call showPoint()
    endIf
    bTrigger=false
    bShowStatus=false
  endIf
end

--- unSelectItem.pgx ---
program unSelectItem()
  local string l_sEvent
  local num i
  local num l_nSize
  local TrajectoryItem l_tTraj
begin
  // remove all the comments
  call trajType:getSizeItem(false,l_nSize)
  for i=0 to (l_nSize-1)
    // get all the items
    call trajType:getTrajItem(l_tTraj,i)
    if find(l_tTraj.comment,"#")!=-1
      // look for the select item
      l_tTraj.comment=right(l_tTraj.comment,len(l_tTraj.comment)-1)
      call trajType:setTrajItem(l_tTraj,i)
    endIf
  endFor
end
